(* Schneider Machine Expert - Basic project tank_level_v9_TM221CE24T, file version 3.0.0.0 *)
(* ProjectInformations: Name=New project *)

HARDWARE
  Cpu 0: TM221CE24T
  ModuleExtensionObject 0: TM3AI4/G
  EthernetConfiguration: NetworkName=M221, IpAllocationMode=FixedAddress, IpAddress=0.0.0.0, SubnetMask=0.0.0.0
  SerialLineConfiguration: Baud=Baud19200, Parity=ParityEven, DataBits=DataBits8, StopBits=StopBits1, PhysicalMedium=PhysicalMediumRs485, TransmissionMode=TransmissionModeModbusRtu, SlaveId=1, Addressing=SlaveAddressing
  MastTask: UsePeriodScanMode=false, PeriodScan=100
  FastTask: Period=255
  CpuBehavior: StartingMode=StartAsPreviousState, AutoSaveRamOnEeprom=true, WatchdogPeriod=250

SYMBOLS  (address, symbol, comment, settings)
  %IW1.0    TANK_LEVEL  [Type=Type_4_20mA, Scope=Scope_Customized, Minimum=300, Maximum=3000]

POU New POU
  (* SectionNumber=0 *)

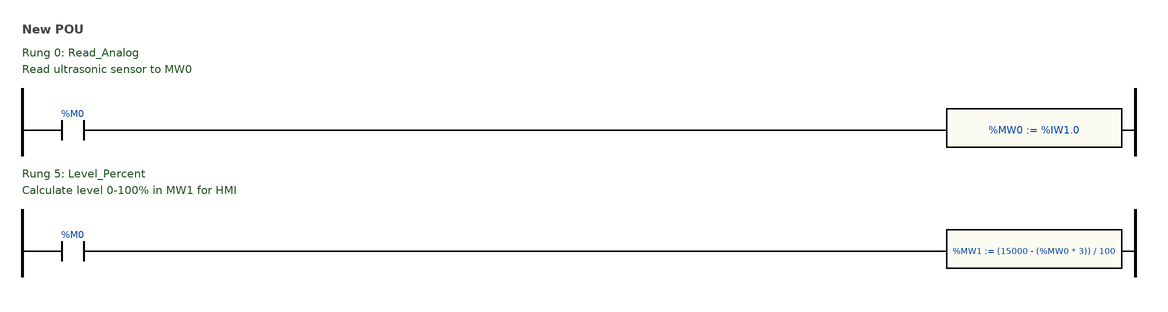

// Rung 0: Read_Analog
// Read ultrasonic sensor to MW0
  LD %M0
  [ %MW0 := %IW1.0 ]      (* TANK_LEVEL *)
  // as ST:
  //   IF %M0 THEN %MW0 := TANK_LEVEL; END_IF;

// Rung 1: Tank_Full_Open_Outlet
// When tank full, SET outlet valve
  LD [%MW0<1800]
  S %Q0.1
  // as ST:
  //   IF %MW0<1800 THEN %Q0.1 := TRUE; END_IF;
  (* the ladder stored for this rung does not match its IL; not drawn *)

// Rung 2: Tank_Empty_Close_Outlet
// When tank empty, RESET outlet valve
  LD [%MW0>4800]
  R %Q0.1
  // as ST:
  //   IF %MW0>4800 THEN %Q0.1 := FALSE; END_IF;
  (* the ladder stored for this rung does not match its IL; not drawn *)

// Rung 3: Tank_Empty_Open_Inlet
// When tank empty, SET inlet valve
  LD [%MW0>4800]
  S %Q0.0
  // as ST:
  //   IF %MW0>4800 THEN %Q0.0 := TRUE; END_IF;
  (* the ladder stored for this rung does not match its IL; not drawn *)

// Rung 4: Tank_Full_Close_Inlet
// When tank full, RESET inlet valve
  LD [%MW0<1800]
  R %Q0.0
  // as ST:
  //   IF %MW0<1800 THEN %Q0.0 := FALSE; END_IF;
  (* the ladder stored for this rung does not match its IL; not drawn *)

// Rung 5: Level_Percent
// Calculate level 0-100% in MW1 for HMI
  LD %M0
  [ %MW1 := (15000 - (%MW0 * 3)) / 100 ]
  // as ST:
  //   IF %M0 THEN %MW1 := (15000 - (%MW0 * 3)) / 100; END_IF;
